PROGRAM p_ModbusRx
VAR
END_VAR

(* Modbus Controls from EPICS *)

(* General System Controls *)
xEnableRemoteControl := mb_Output_Coils[0];
g_xEstop		:= mb_Output_Coils[1];

IF xEnableRemoteControl THEN
xN2Purge	:= mb_Output_Coils[9];

(* Selector Controls *)
stSelector.iVici1ReqPos := mb_Output_Registers[30];
stSelector.iVici2ReqPos := mb_Output_Registers[31];
stSelector.iSyncReqPos	:= mb_Output_Registers[32];

stSelector.xResLock := mb_Output_Coils[30];
stSelector.xFMReset := mb_Output_Coils[31];
stSelector.xFMModeReq 	:= mb_Output_Coils[32];
stSelector.xResUnlock := mb_Output_Coils[33];

stSelector.stShaker01.i_xEpics := mb_Output_Coils[10];
stSelector.stShaker02.i_xEpics := mb_Output_Coils[11];
stSelector.stShaker03.i_xEpics := mb_Output_Coils[12];
stSelector.stShaker04.i_xEpics := mb_Output_Coils[13];

(* Selector 2 Controls *)
stSelector2.iVici1ReqPos := mb_Output_Registers[40];
stSelector2.iVici2ReqPos := mb_Output_Registers[41];
stSelector2.iSyncReqPos	:= mb_Output_Registers[42];

stSelector2.xResLock := mb_Output_Coils[40];
stSelector2.xFMReset := mb_Output_Coils[41];
stSelector2.xFMModeReq 	:= mb_Output_Coils[42];
stSelector2.xResUnlock := mb_Output_Coils[43];

stSelector2.stShaker01.i_xEpics := mb_Output_Coils[44];
stSelector2.stShaker02.i_xEpics := mb_Output_Coils[45];
stSelector2.stShaker03.i_xEpics := mb_Output_Coils[46];
stSelector2.stShaker04.i_xEpics := mb_Output_Coils[47];

(* Proportionair controls *)
stRegProp1.xEnable:=mb_Output_Coils[50];  //Proportionair controls
stRegProp2.xEnable:=mb_Output_Coils[51];  //Proportionair controls

stRegProp3.xEnable:=mb_Output_Coils[52];  //Proportionair controls
stRegProp4.xEnable:=mb_Output_Coils[53];  //Proportionair controls

stRegProp1.iSetpoint:=mb_Output_Registers[50];  //Proportionair controls
stRegProp2.iSetpoint:=mb_Output_Registers[51];  //Proportionair controls
stRegProp1.iHiLimit:=mb_Output_Registers[52];  //Proportionair controls
stRegProp2.iHiLimit:=mb_Output_Registers[53];  //Proportionair controls

stRegProp3.iSetpoint:=mb_Output_Registers[54];  //Proportionair controls
stRegProp4.iSetpoint:=mb_Output_Registers[55];  //Proportionair controls
stRegProp3.iHiLimit:=mb_Output_Registers[56];  //Proportionair controls
stRegProp4.iHiLimit:=mb_Output_Registers[57];  //Proportionair controls

(* Digital output controls *)
stGasMani.stManiVlv1.xSW:=mb_Output_Coils[60];  //Minitti manifold valve controls
stGasMani.stManiVlv2.xSW:=mb_Output_Coils[61];  //Minitti manifold valve controls
stGasMani.stManiVlv3.xSW:=mb_Output_Coils[62];  //Minitti manifold valve controls
stGasMani.stManiVlv4.xSW:=mb_Output_Coils[63];  //Minitti manifold valve controls
stGasMani.stManiVlv5.xSW:=mb_Output_Coils[64];  //Minitti manifold valve controls
stGasMani.stManiVlv6.xSW:=mb_Output_Coils[65];  //Minitti manifold valve controls
stGasMani.stManiVlv7.xSW:=mb_Output_Coils[66];  //Minitti manifold valve controls
stGasMani.stManiVlv8.xSW:=mb_Output_Coils[67];  //Minitti manifold valve controls
//=========================================================
// ALI Controls
	stALI.axisX.xStart:=mb_Output_Coils[80];  //ALI_Manip
	stALI.axisX.xStop:=mb_Output_Coils[81];  //ALI_Manip
	stALI.axisY.xStart:=mb_Output_Coils[82];  //ALI_Manip
	stALI.axisY.xStop:=mb_Output_Coils[83];  //ALI_Manip
	stALI.axisZ.xStart:=mb_Output_Coils[84];  //ALI_Manip
	stALI.axisZ.xStop:=mb_Output_Coils[85];  //ALI_Manip
	
	stALI.stPropVlv.xEnable := mb_Output_Coils[86];
	
	stALI.axisX.xReset:=mb_Output_Coils[87];  //ALI_Manip
	stALI.axisY.xReset:=mb_Output_Coils[88];  //ALI_Manip
	stALI.axisZ.xReset:=mb_Output_Coils[89];  //ALI_Manip
	
	stALI.stPropVlv.i_iPercOpenSP := mb_Output_Registers[80]; //ALI Propvalve
	stALI.stPropVlv.ePVCtrlStateReq := mb_Output_Registers[81]; //ALI Propvalve
	MEMCPY(srcAddr:=ADR(mb_PLC_Memory[90]), destAddr:=ADR(stALI.axisX.rReqAbsPos), n:=SIZEOF(stALI.axisX.rReqAbsPos)); //ALI CTRL
	MEMCPY(srcAddr:=ADR(mb_PLC_Memory[92]), destAddr:=ADR(stALI.axisY.rReqAbsPos), n:=SIZEOF(stALI.axisY.rReqAbsPos)); //ALI CTRL
	MEMCPY(srcAddr:=ADR(mb_PLC_Memory[94]), destAddr:=ADR(stALI.axisZ.rReqAbsPos), n:=SIZEOF(stALI.axisZ.rReqAbsPos)); //ALI CTRL
	MEMCPY(srcAddr:=ADR(mb_PLC_Memory[96]), destAddr:=ADR(stALI.stPropVlv.i_rPressSP), n:=SIZEOF(stALI.stPropVlv.i_rPressSP)); //ALI CTRL

END_IF

END_PROGRAM

(* stored: Version 1.1.0.1, ProductVersion 3.1.4020.12
   POU p_ModbusRx: Id {20750476-3750-4dd9-9eaa-26d5f7c2ab85}, SpecialFunc None *)
